Yaskawa INFORM job: R2_W30(0,0)_MP_OK.JBI

/JOB
//NAME R2_W30(0,0)_MP_OK
///FOLDERNAME MP_TEST
//POS
///NPOS 41,41,0,2,0,0
///TOOL 0
///POSTYPE PULSE
///PULSE
C00000=134519,-57362,-86948,-86332,82118,-51299
C00001=134414,-57361,-91245,-85703,76372,-52551
C00002=72543,-54297,-24085,-64724,83626,-76847
C00003=68475,-56773,-25387,-65356,80829,-77250
C00004=66794,-57679,-25855,-65610,79679,-77420
C00005=66871,-58906,-26483,-65635,79622,-77306
C00006=65370,-58650,-26352,-65830,78686,-77544
C00007=66871,-58906,-26483,-65635,79622,-77306
C00008=66794,-57679,-25855,-65610,79679,-77420
C00009=66304,-46286,-19628,-71230,87881,-79359
C00010=66333,-46854,-19955,-71226,87869,-79316
C00011=66304,-46286,-19628,-71230,87881,-79359
C00012=69376,-46935,-20004,-70733,89901,-78956
C00013=61359,-70402,-31957,-61472,66977,-76524
C00014=48122,-68303,-31001,-61838,59163,-79107
C00015=47009,-69217,-31415,-61960,58378,-79212
C00016=48122,-68303,-31001,-61838,59163,-79107
C00017=61359,-70402,-31957,-61472,66977,-76524
C00018=61697,-68561,-31129,-61292,67400,-76654
C00019=63542,-68103,-30922,-61115,68573,-76378
C00020=68063,-66735,-30294,-60626,71468,-75723
C00021=43897,-38871,7150,-70138,78370,-46376
C00022=40267,-40033,6474,-71163,76059,-46702
C00023=38986,-41072,6113,-71581,75157,-46704
C00024=38647,-41357,4222,-71434,75295,-47194
C00025=40101,-39394,7145,-71227,75927,-46683
C00026=39200,-40646,6795,-71567,75222,-46588
C00027=40051,-39411,6837,-71201,75959,-46769
C00028=46280,-34439,9818,-69383,80077,-46377
C00029=66285,-44840,3736,-66754,79755,-29237
C00030=62767,-44916,3697,-67757,77640,-29677
C00031=61360,-44896,3709,-68148,76793,-29854
C00032=61352,-45632,1832,-67999,77097,-30192
C00033=62907,-45297,3395,-67719,77720,-29656
C00034=61959,-41523,5595,-67864,77383,-30028
C00035=63033,-34718,9629,-67397,78445,-30330
C00036=63526,-31211,11825,-67204,78931,-30459
C00037=64746,-31188,11839,-66885,79675,-30302
C00038=67791,-31012,11948,-66069,81530,-29909
C00039=94001,-97744,-45654,-30172,80481,-23781
C00040=134519,-57362,-86948,-86332,82118,-51299
BC00000=15,15,1063921
BC00001=15,15,102776
BC00002=15,0,583436
BC00003=15,0,572372
BC00004=15,0,567947
BC00005=15,0,551042
BC00006=15,0,550553
BC00007=15,0,551042
BC00008=15,0,567947
BC00009=15,0,520815
BC00010=15,0,513082
BC00011=15,0,520815
BC00012=15,0,522121
BC00013=15,0,609559
BC00014=4565,0,603345
BC00015=3340,0,605584
BC00016=4565,0,603345
BC00017=15,0,609559
BC00018=15,0,607303
BC00019=15,0,613094
BC00020=15,0,627570
BC00021=15,-36082,720158
BC00022=15,-36082,702643
BC00023=15,-36082,695637
BC00024=15,-36082,695637
BC00025=15,-36082,695637
BC00026=18859,-36082,682029
BC00027=18164,-36082,689035
BC00028=16886,-36082,693512
BC00029=15,0,740175
BC00030=15,0,720225
BC00031=15,0,712245
BC00032=15,0,712245
BC00033=15,0,712245
BC00034=15,0,707815
BC00035=15,0,698952
BC00036=15,0,694424
BC00037=15,0,702404
BC00038=15,0,722354
BC00039=15,0,722354
BC00040=15,217251,1063921
///POSTYPE BASE
///RECTAN
///RCONF 0,0,0,0,0,0,0,0,0,0,0,0,0,0,0,0,0,0,0,0,0,0,0,0
P00006=0.222,-3.123,-1.508,0.0000,0.0000,0.0000
P00022=0.222,-3.123,-1.508,0.0000,0.0000,0.0000
//INST
///DATE 2023/11/16 10:45
///ATTR SC,RW
///GROUP1 RB1,BS1
NOP
'r2_W30(0,0)
JUMP *LABEL
'Path VIA934
SFTOF
MOVJ C00000 BC00000 VJ=20.00
'Path VIA935
SFTOF
MOVJ C00001 BC00001 VJ=20.00
COMM 'Path S936
COMM SFTOF
COMM MOVJ C00002 BC00002 VJ=100.00
COMM MOVJ C00003 BC00003 VJ=100.00
COMM MOVL C00004 BC00004 V=100.0
COMM MOVL C00005 BC00005 V=60.0
COMM REFP 3 C00006 BC00006
COMM CALL JOB:SEARCH-R1
COMM SET P022 P006
COMM SFTON P022
COMM MOVL C00007 BC00007 V=60.0
COMM MOVL C00008 BC00008 V=100.0
COMM MOVL C00009 BC00009 V=60.0
COMM REFP 3 C00010 BC00010
COMM CALL JOB:SEARCH-R1
COMM SET P022 P006
COMM SFTON P022
COMM MOVL C00011 BC00011 V=60.0
COMM MOVL C00012 BC00012 V=100.0
COMM MOVL C00013 BC00013 V=100.0
COMM MOVL C00014 BC00014 V=60.0
COMM REFP 3 C00015 BC00015
COMM CALL JOB:SEARCH-R1
COMM SET P022 P006
COMM SFTON P022
COMM MOVL C00016 BC00016 V=60.0
COMM MOVL C00017 BC00017 V=100.0
COMM MOVL C00018 BC00018 V=100.0
COMM MOVL C00019 BC00019 V=400.0
COMM MOVL C00020 BC00020 V=1000.0
COMM 'Path W937
COMM SFTOF
COMM SFTON P022
COMM MOVJ C00021 BC00021 VJ=100.00
COMM MOVJ C00022 BC00022 VJ=100.00
COMM MOVL C00023 BC00023 V=100.0 PL=0
COMM REFP 1 C00024 BC00024
COMM REFP 2 C00025 BC00025
COMM MACRO1 MJ#(0) ARGF7
COMM ARCON
COMM MOVL C00026 BC00026 V=11.7
COMM ARCOF
COMM MOVL C00027 BC00027 V=400.0
COMM MOVL C00028 BC00028 V=1000.0
COMM SFTOF
COMM 'Path W938
COMM SFTOF
COMM SFTON P022
COMM MOVJ C00029 BC00029 VJ=100.00
COMM MOVJ C00030 BC00030 VJ=100.00
COMM MOVL C00031 BC00031 V=100.0 PL=0
COMM REFP 1 C00032 BC00032
COMM REFP 2 C00033 BC00033
COMM MACRO1 MJ#(0) ARGF7
COMM ARCON
COMM MOVL C00034 BC00034 V=11.7
COMM MOVL C00035 BC00035 V=11.7
COMM MOVL C00036 BC00036 V=11.7
COMM ARCOF
COMM MOVL C00037 BC00037 V=400.0
MOVL C00038 BC00038 V=100.0
MOVJ C00039 BC00039 VJ=20.00
MOVJ C00040 BC00040 VJ=20.00
SFTOF
*LABEL
END
